TEXTLIST TextList_TwinSAFE_FB_ESTOP_State
  0 = 'undefined'
  1 = 'RUN'
  2 = 'STOP'
  3 = 'SAFE'
  4 = 'ERROR'
  5 = 'RESET'
  6 = 'START'
  8 = 'DELAYOUT'
   = ''
END_TEXTLIST

(* stored: Version 1.1.0.1, ProductVersion 3.1.4024.11
   TextList TextList_TwinSAFE_FB_ESTOP_State: Id {43822800-fde2-4daf-b607-53ce430cfedd} *)
